INTERFACE I_Focus EXTENDS I_BaseAxis

END_INTERFACE

(* stored: Version 1.1.0.1, ProductVersion 3.1.4026.11
   Itf I_Focus: Id {1a3f6670-f8af-4019-b502-f4da4afb4275} *)
